(* CODESYS project Apollo_001_V1_CleanLease_Gemert_RECOVERED_2025-04-10T15-18-59.project

Project tree, tasks and I/O mapping:
  Device : CPX-E-CEC-M1-PN, Festo, order no. 4252743, version 3.5.16.46
    application Application
      libraries: Standard, 3.5.15.0 (System); CmpOPCUAClient, 3.5.17.0 (System); CmpOPCUAStack, 3.5.17.0 (System); IecVarAccessOpcUaMetaData Interfaces, * (System); CmpOPCUAServer Interfaces, * (System); Datasource OpcUa, * (3S - Smart Software Solutions GmbH); IecVarAccess3 Interfaces, * (System); SymbolicVarsBase, 3.5.16.30 (System); CmpBitmapPool, * (System)
      task MainTask (cyclic, interval t#20ms, priority 20) calls nothing
      task VISU_TASK (cyclic, interval 100 ms, priority 31) calls VisuElems.Visu_Prg
      task EtherCAT_Task (cyclic, interval t#8ms, priority 1) calls Apollo_Test_Mode, Apollo_Machine_State_V2, Set_Parameter_Prog, Test_Full_Prod, Dropconveyor
      program PLC_PRG [ST]
      image pool ImagePool
      Symbols
      Old_Progs/
        program Apollo_Machine_State [ST]
        function block FunctionBlock_Move_Guiders_Apollo [ST]
        program Apollo_Running_Guiders_AND_PickConveyor [ST]
        function block FunctionBlock_Move_Conveyor_Drop [ST]
        program Apollo_Running_GuiderMovement [ST]
      Progs_In_Apollo/
        Test_Mode/
          program Apollo_Test_Mode [ST]
          program Test_Full_Prod [ST]
        Machine State/
          program Set_Parameter_Prog [ST]
          program Apollo_Machine_State_V2 [ST]
        Run_Mode/
        FunctionBlocks/
          function block FunctionBlock_Gripper_Drop [ST]
          function block FunctionBlock_Move_To_Pos [ST]
          function block FunctionBlock_Gripper_Grip [ST]
          function block FunctionBlock_Activate_Ventilator [ST]
          function block FunctionBlock_Move_Pick_Conveyor [ST]
      visualisation Main_Page
      Variables_AND_Parameters/
        global variables Parameters
        global variables GVL_1
      Prog_In_DEV/
        Function Blocks/
        Programms/
          program Dropconveyor [ST]
          program Apollo_RunMode_Main [ST]
    SoftMotion General Axis Pool
    PLC_Diagnosis : PLC-Diagnosis, Festo AG & Co. KG, version 3.5.4.4
    CPX_E_System : CPX_E_System, Festo, order no. 4252743, version 1.311
      E_4AO_U_I : E-4AO-U-I, Festo, order no. 4080494, version 1.311
          settings:  = 0;  = 1;  = 1;  = 1;  = 1;  = 0;  = 0;  = 1;  = 144;  = 144;  = 144;  = 144;  = 1;  = 1;  = 1;  = 1;  = 0;  = 0;  = 0;  = 0;  = 0;  = 0;  = 0;  = 0;  = 0;  = 0;  = 0;  = 0;  = 0;  = 0;  = 0;  = 0;  = 0;  = 0;  = 0;  = 0;  = 0;  = 0;  = 0;  = 0;
             = 4466775293954;  = 'PI%i.0.1.1=1';  = 'PI%i.0.2.1=1';  = 'PI%i.0.7.1=1';  = 'PI%i.1.1.1=1';  = 'PI%i.1.3.1=0';  = 'PI%i.6.0.1=0';  = 'PI%i.6.5.1=1';  = 'PI%i.7.0.8=144';  = 'PI%i.8.0.8=144';  = 'PI%i.9.0.8=144';  = 'PI%i.10.0.8=144';  = 'PI%i.11.0.4=1';  = 'PI%i.11.4.4=1';  = 'PI%i.12.0.4=1';  = 'PI%i.12.4.4=1';  = dd8ed08c;  = 2
          output Application.GVL_1.Ventilator : UINT  // Output 0
          unmapped channels: Output 1, Output 2, Output 3
      E_8DO : E-8DO, Festo, order no. 4080491, version 1.311
          settings:  = 0;  = 1;  = 1;  = 0;  = 0;  = 0;  = 0;  = 0;  = 0;  = 0;  = 0;  = 0;  = 0;  = 0;  = 0;  = 0;  = 0;  = 0;  = 0;  = 0;  = 0;  = 0;  = 0;  = 0;  = 0;  = 0;  = 0;  = 0;  = 0;  = 0;  = 0;  = 0;  = 0;  = 0;  = 0;  = 0;  = 0;  = 0;  = 0;  = 0;
             = 0;  = 0;  = 0;  = 0;  = 0;  = 0;  = 0;  = 0;  = 0;  = 0;  = 0;  = 0;  = 8800390021120;  = 'PI%i.0.1.1=1';  = 'PI%i.0.2.1=1';  = 'PI%i.1.1.1=0';  = dd8aeb00;  = 1
          output Application.GVL_1.Conveyor_Pick_Speed_A : BOOL  // Output 0.Bit0
          output Application.GVL_1.Conveyor_Pick_Speed_B : BOOL  // Output 0.Bit1
          output Application.GVL_1.Conveyor_Pick_Speed_C : BOOL  // Output 0.Bit2
          output Application.GVL_1.Conveyor_Pick_Reverse : BOOL  // Output 0.Bit3
          output Application.GVL_1.Conveyor_Drop_Speed_A : BOOL  // Output 0.Bit4
          output Application.GVL_1.Conveyor_Drop_Speed_B : BOOL  // Output 0.Bit5
          output Application.GVL_1.Conveyor_Drop_Speed_C : BOOL  // Output 0.Bit6
          output Application.GVL_1.Conveyor_Drop_Reverse : BOOL  // Output 0.Bit7
          unmapped channels: Output 0
      E_8DO_1 : E-8DO, Festo, order no. 4080491, version 1.311
          settings:  = 0;  = 1;  = 1;  = 0;  = 0;  = 0;  = 0;  = 0;  = 0;  = 0;  = 0;  = 0;  = 0;  = 0;  = 0;  = 0;  = 0;  = 0;  = 0;  = 0;  = 0;  = 0;  = 0;  = 0;  = 0;  = 0;  = 0;  = 0;  = 0;  = 0;  = 0;  = 0;  = 0;  = 0;  = 0;  = 0;  = 0;  = 0;  = 0;  = 0;
             = 0;  = 0;  = 0;  = 0;  = 0;  = 0;  = 0;  = 0;  = 0;  = 0;  = 0;  = 0;  = 8800390021120;  = 'PI%i.0.1.1=1';  = 'PI%i.0.2.1=1';  = 'PI%i.1.1.1=0';  = dd8b5e24;  = 1
          output Application.GVL_1.Gripper : BOOL  // Output 0.Bit0
          output Application.GVL_1.Blow_Out : BOOL  // Output 0.Bit1
          output Application.GVL_1.VacuumBlow : BOOL  // Output 0.Bit2
          unmapped channels: Output 0
      E_16DI : E-16DI, Festo, order no. 4080492, version 1.311
          settings:  = 0;  = 1;  = 1;  = 1;  = 1;  = 0;  = 0;  = 0;  = 0;  = 0;  = 0;  = 0;  = 0;  = 0;  = 0;  = 0;  = 0;  = 0;  = 0;  = 0;  = 0;  = 0;  = 0;  = 0;  = 0;  = 0;  = 0;  = 0;  = 0;  = 0;  = 0;  = 0;  = 0;  = 0;  = 0;  = 0;  = 0;  = 0;  = 0;  = 0;
             = 0;  = 0;  = 0;  = 0;  = 0;  = 0;  = 0;  = 0;  = 0;  = 0;  = 0;  = 0;  = 0;  = 1153202979585458176;  = 'PI%i.0.0.1=1';  = 'PI%i.1.0.1=1';  = 'PI%i.1.4.2=1';  = 'PI%i.1.6.2=1';  = 'PI%i.6.0.1=0';  = 'PI%i.6.1.1=0';  = 'PI%i.6.2.1=0';  = 'PI%i.6.3.1=0';  = 'PI%i.6.4.1=0';  = 'PI%i.6.5.1=0';  = 'PI%i.6.6.1=0';  = 'PI%i.6.7.1=0';  = 'PI%i.7.0.1=0';  = 'PI%i.7.1.1=0';  = 'PI%i.7.2.1=0';  = 'PI%i.7.3.1=0';  = 'PI%i.7.4.1=0';  = 'PI%i.7.5.1=0';  = 'PI%i.7.6.1=0';  = 'PI%i.7.7.1=0';  = dd8b6c92;  = 1
          input  Application.GVL_1.PHC_PickConveyor_END : BOOL  // Input 0.Bit0
          input  Application.GVL_1.Start_production_Button : BOOL  // Input 0.Bit2
          input  Application.GVL_1.PHC_Drop_Conveyor : BOOL  // Input 0.Bit6
          unmapped channels: Input 0
      E_CEC_M1_PN : E-CEC-M1-PN, Festo, order no. 4252743, version 1.311
          settings:  = 0;  = 15365580000768;  = 16820416;  = 16777215;  = 0;  = 14549093;  = 1f93f90d;  = 11
    PROFINET_Device : PROFINET Device, Festo, version 3.5.15.2
    EtherCAT_Master : EtherCAT Master, Festo, version 3.5.16.43
      CMMT_AS_MP_S1 : CMMT-AS-MP-S1 (SoftMotion), Festo, order no. 814316x, version 4.0.33.0
          settings: StationAlias = 0
          unmapped channels: Controlword, Modes of operation, Target position, Profile velocity, Target velocity, Target torque, Velocity offset, Torque offset, Touch probe function, ---, Statusword, Modes of operation display, Position actual value, Velocity actual value, Torque actual value, Touch probe status, Touch probe 1 positive edge, Touch probe 1 negative edge, Touch probe 2 positive edge, Touch probe 2 negative edge, ---
        Inner_Rail : SM_Drive_EtherCAT_Festo_CMMT_AS_MP_S1, Festo, version 4.0.33.0
            settings: wDriveID = 0; fSWLimitPositive = 1400; fSWLimitNegative = -50; AdrOffset_8010 = 12; BitOffset_8010 = 0; BitLength_8010 = 16; Address_8010 = '%QW6'; Type_8010 = 'UINT'; AddressPointer_8010 = ADR(%QW6); AdrOffset_8020 = 14; BitOffset_8020 = 0; BitLength_8020 = 8; Address_8020 = '%QB14'; Type_8020 = 'SINT'; AddressPointer_8020 = ADR(%QB14); AdrOffset_8030 = 16; BitOffset_8030 = 0; BitLength_8030 = 32; Address_8030 = '%QD4'; Type_8030 = 'DINT'; AddressPointer_8030 = ADR(%QD4); AdrOffset_8040 = 24; BitOffset_8040 = 0; BitLength_8040 = 32; Address_8040 = '%QD6'; Type_8040 = 'DINT'; AddressPointer_8040 = ADR(%QD6); AdrOffset_8050 = 28; BitOffset_8050 = 0; BitLength_8050 = 16; Address_8050 = '%QW14'; Type_8050 = 'INT'; AddressPointer_8050 = ADR(%QW14); AdrOffset_8060 = 38; BitOffset_8060 = 0; BitLength_8060 = 16; Address_8060 = '%QW19'; Type_8060 = 'UINT'; AddressPointer_8060 = ADR(%QW19); AdrOffset_8510 = 4;
              BitOffset_8510 = 0; BitLength_8510 = 16; Address_8510 = '%IW2'; Type_8510 = 'UINT'; AddressPointer_8510 = ADR(%IW2); AdrOffset_8520 = 6; BitOffset_8520 = 0; BitLength_8520 = 8; Address_8520 = '%IB6'; Type_8520 = 'SINT'; AddressPointer_8520 = ADR(%IB6); AdrOffset_8530 = 8; BitOffset_8530 = 0; BitLength_8530 = 32; Address_8530 = '%ID2'; Type_8530 = 'DINT'; AddressPointer_8530 = ADR(%ID2); AdrOffset_8540 = 12; BitOffset_8540 = 0; BitLength_8540 = 32; Address_8540 = '%ID3'; Type_8540 = 'DINT'; AddressPointer_8540 = ADR(%ID3); AdrOffset_8550 = 16; BitOffset_8550 = 0; BitLength_8550 = 16; Address_8550 = '%IW8'; Type_8550 = 'INT'; AddressPointer_8550 = ADR(%IW8); AdrOffset_8560 = 18; BitOffset_8560 = 0; BitLength_8560 = 16; Address_8560 = '%IW9'; Type_8560 = 'UINT'; AddressPointer_8560 = ADR(%IW9); AdrOffset_8570 = 20; BitOffset_8570 = 0; BitLength_8570 = 32; Address_8570 = '%ID5'; Type_8570 = 'DINT';
              AddressPointer_8570 = ADR(%ID5); AdrOffset_8580 = 24; BitOffset_8580 = 0; BitLength_8580 = 32; Address_8580 = '%ID6'; Type_8580 = 'DINT'; AddressPointer_8580 = ADR(%ID6); AdrOffset_8590 = 28; BitOffset_8590 = 0; BitLength_8590 = 32; Address_8590 = '%ID7'; Type_8590 = 'DINT'; AddressPointer_8590 = ADR(%ID7); AdrOffset_8600 = 32; BitOffset_8600 = 0; BitLength_8600 = 32; Address_8600 = '%ID8'; Type_8600 = 'DINT'; AddressPointer_8600 = ADR(%ID8)
      CMMT_AS_MP_S1_1 : CMMT-AS-MP-S1 (SoftMotion), Festo, order no. 814316x, version 4.0.33.0
          settings: StationAlias = 0
          unmapped channels: Controlword, Modes of operation, Target position, Profile velocity, Target velocity, Target torque, Velocity offset, Torque offset, Touch probe function, ---, Statusword, Modes of operation display, Position actual value, Velocity actual value, Torque actual value, Touch probe status, Touch probe 1 positive edge, Touch probe 1 negative edge, Touch probe 2 positive edge, Touch probe 2 negative edge, ---
        Outer_Rail : SM_Drive_EtherCAT_Festo_CMMT_AS_MP_S1, Festo, version 4.0.33.0
            settings: fSWLimitPositive = 1400; fSWLimitNegative = -50; AdrOffset_8010 = 44; BitOffset_8010 = 0; BitLength_8010 = 16; Address_8010 = '%QW22'; Type_8010 = 'UINT'; AddressPointer_8010 = ADR(%QW22); AdrOffset_8020 = 46; BitOffset_8020 = 0; BitLength_8020 = 8; Address_8020 = '%QB46'; Type_8020 = 'SINT'; AddressPointer_8020 = ADR(%QB46); AdrOffset_8030 = 48; BitOffset_8030 = 0; BitLength_8030 = 32; Address_8030 = '%QD12'; Type_8030 = 'DINT'; AddressPointer_8030 = ADR(%QD12); AdrOffset_8040 = 56; BitOffset_8040 = 0; BitLength_8040 = 32; Address_8040 = '%QD14'; Type_8040 = 'DINT'; AddressPointer_8040 = ADR(%QD14); AdrOffset_8050 = 60; BitOffset_8050 = 0; BitLength_8050 = 16; Address_8050 = '%QW30'; Type_8050 = 'INT'; AddressPointer_8050 = ADR(%QW30); AdrOffset_8060 = 70; BitOffset_8060 = 0; BitLength_8060 = 16; Address_8060 = '%QW35'; Type_8060 = 'UINT'; AddressPointer_8060 = ADR(%QW35); AdrOffset_8510 = 40; BitOffset_8510 = 0;
              BitLength_8510 = 16; Address_8510 = '%IW20'; Type_8510 = 'UINT'; AddressPointer_8510 = ADR(%IW20); AdrOffset_8520 = 42; BitOffset_8520 = 0; BitLength_8520 = 8; Address_8520 = '%IB42'; Type_8520 = 'SINT'; AddressPointer_8520 = ADR(%IB42); AdrOffset_8530 = 44; BitOffset_8530 = 0; BitLength_8530 = 32; Address_8530 = '%ID11'; Type_8530 = 'DINT'; AddressPointer_8530 = ADR(%ID11); AdrOffset_8540 = 48; BitOffset_8540 = 0; BitLength_8540 = 32; Address_8540 = '%ID12'; Type_8540 = 'DINT'; AddressPointer_8540 = ADR(%ID12); AdrOffset_8550 = 52; BitOffset_8550 = 0; BitLength_8550 = 16; Address_8550 = '%IW26'; Type_8550 = 'INT'; AddressPointer_8550 = ADR(%IW26); AdrOffset_8560 = 54; BitOffset_8560 = 0; BitLength_8560 = 16; Address_8560 = '%IW27'; Type_8560 = 'UINT'; AddressPointer_8560 = ADR(%IW27); AdrOffset_8570 = 56; BitOffset_8570 = 0; BitLength_8570 = 32; Address_8570 = '%ID14'; Type_8570 = 'DINT'; AddressPointer_8570 = ADR(%ID14);
              AdrOffset_8580 = 60; BitOffset_8580 = 0; BitLength_8580 = 32; Address_8580 = '%ID15'; Type_8580 = 'DINT'; AddressPointer_8580 = ADR(%ID15); AdrOffset_8590 = 64; BitOffset_8590 = 0; BitLength_8590 = 32; Address_8590 = '%ID16'; Type_8590 = 'DINT'; AddressPointer_8590 = ADR(%ID16); AdrOffset_8600 = 68; BitOffset_8600 = 0; BitLength_8600 = 32; Address_8600 = '%ID17'; Type_8600 = 'DINT'; AddressPointer_8600 = ADR(%ID17)
  libraries: VisuSymbols, 4.5.0.0 (System)
  5ce3da45-db07-42e7-a21c-a00fff4ed8f6|C:\Users\RobinvanNieuwenhuyse\Downloads\Landuwasco-logo.png
  text list GlobalTextList
*)

// Device/Application/Variables_AND_Parameters/Parameters
{attribute 'qualified_only'}
VAR_GLOBAL PERSISTENT RETAIN
//-------------------------------------------------------------------------------------------------
//Positions
	//Readypos
	ReadyPos_Inner:INT;
	ReadyPos_Outer:INT;
	
	//Pick_Pos
	Pick_Pos_Inner_Test_Prod:INT;
	Pick_Pos_Outer_Test_Prod:INT;
	
	//Drop_Pos
	Drop_Pos_Inner:INT;
	Drop_Pos_Outer:INT;
	
	Drop_Pos_Inner_Test_Prod:INT;
	Drop_Pos_Outer_Test_Prod:INT;
	
	//Before Drop Pos
	Before_Drop_Pos_Inner:INT;
	Before_Drop_Pos_Outer:INT;
	
	//Distances
	Distance_Move_After_PHC:LREAL; // distance in mm
	
	
	//Points between readypos and Pick_Pos called RPP_CheckPointPos
	
//-------------------------------------------------------------------------------------------------
//Dynamics
	//Test 
	Speed_Test_Prod:LREAL; // for the test production cycly
	ACC_DEC_Test_Prod:LREAl;
	Jerk_Test_Prod:LREAL;
	
	Speed_Test_Prod_Slow:LREAL;
	ACC_DEC_Test_Prod_Slow:LREAL;
	Jerk_Test_prod_Slow:LREAL;
	
	//Production
	Vel_Prod:LREAL;
	Acc_Dec_Prod:LREAL;
	Jerk_Prod:LREAL;
//-------------------------------------------------------------------------------------------------
//Timers

//Wait times
	Wait_Time_NoBatch:INT;	
	Wait_Time_Piece_Drop_Conveyor:INT;// max time the drop conveyor can run (if no pieces are detected
	Wait_Time_AI:INT;
	
//Delays
	Delay_Gripper_Closed_Before_Moving:INT;
	Delay_Move_After_Piece_Dropped:INT;
	Delay_Blow_Vacuum:INT;
	Delay_Move_Conveyor_After_PHC_Covered:INT;
	Delay_DropBox_Opened:INT;
	Delay_Conveyor_Move_After_DropBox_Opened:INT;
	Delay_Gripper_Open_During_Drop:INT;
//-------------------------------------------------------------------------------------------------
// Settings
	//Ventilator
	Ventilator_Strength:INT;	

	//Conveyors
	Conveyor_Speed_Pick:INT;	
	Conveyor_Speed_Drop:INT;		

	Delay_Blow:INT;

END_VAR

// Device/Application/Variables_AND_Parameters/GVL_1
{attribute 'qualified_only'}
VAR_GLOBAL
//-------------------------------------------------------------------------------------------------	
// AI 
	//States
	AI_Start:BOOL;
	AI_Done:BOOL;
	AI_Detection_Memory:BOOL;
	
	AI_USE_TestProd:BOOL;
	
	//Detections
	Pick_Pos_Inner:INT;
	Pick_Pos_Outer:INT;
	
	Conveyor_Pick_Move_Left:BOOL;
	Conveyor_Pick_Move_Right:BOOL;
	Conveyor_Pick_Time:INT; // Time in ms for movement left or right
	Conveyor_Movement_Memory:BOOL; // check if conveyor already moved due to detections before
//-------------------------------------------------------------------------------------------------		
// Robot Command Settings

	//Power Drives
	Power_Drive_InnerRail:MC_Power;
	Power_Drive_OuterRail:MC_Power;
	
	//Reset
	Reset_InnerRail:MC_Reset;
	Reset_OuterRail:MC_Reset;
	
	//movements 
	Move_To_Pos_InnerRail:MC_MoveAbsolute;
	Move_To_Pos_OuterRail:MC_MoveAbsolute;
	
	//Stop movement and set axis in standstill
	Halt_Inner:MC_Halt;
	Halt_Outer:MC_Halt;
//-------------------------------------------------------------------------------------------------		
//	Buttons
	Turn_On:BOOL; // OPCUA communicated
	Turn_Off:BOOL; // OPCUA communicated
	Reset:BOOL;
	Start_production_Button:BOOL;
//-------------------------------------------------------------------------------------------------	
//Sensors
	//PHC
	PHC_PickConveyor_Front:BOOL; //first PHC in cycle picking
	PHC_PickConveyor_END:BOOL;  // last PHC
	
	
	PHC_Reach_Batch:BOOL;
	PHC_Drop_Conveyor:BOOL;
	PHC_Gripper:BOOL;
//-------------------------------------------------------------------------------------------------	
//Actuators

	//Conveyors
	Conveyor_Pick_Speed_A:BOOL;
	Conveyor_Pick_Speed_B:BOOL;
	Conveyor_Pick_Speed_C:BOOL;
	Conveyor_Pick_Reverse:BOOL;
	Test_Conveyor_Pick_Choose_Speed:INT:=1;
	
	Conveyor_Drop_Speed_A:BOOL;
	Conveyor_Drop_Speed_B:BOOL;
	Conveyor_Drop_Speed_C:BOOL;
	Conveyor_Drop_Reverse:BOOL;
	Test_coveyor_Drop_Choos_Speed:INT:=1;
	
	//Gripper
	Gripper:BOOL;
	VacuumBlow:BOOL;
	Blow_Out:BOOL;
	
	//Ventilator
	Ventilator:INT;
	
	//DropBox
	Cylinder_DropBox:BOOL;
	
//-------------------------------------------------------------------------------------------------	
// State of Robot
//Positions
	//Current Pos
	Current_Pos_Inner:LREAL;
	Current_Pos_Outer:LREAL;
// Cases of Robot
	//Test
	enStepTestProd:INT; // this variable is purely to test prod during dev
	enStepTest:INT; //case for testmode

	
	//Prod
	enStepBoot:INT; // case int for bootup proces
	enStepRun:INT; // case int for when robot is running
	enStepRunMove:INT; //case int for moving robot
	enStepDrop:INT;
	
//Cases of Functions
	enFBMoveGuider:INT; // case int for certain movements
	enFBMoveConveyor_Pick:INT;
	enFBMoveConveyor_Drop:INT;
	enFBGripping:INT;
	enFBDropping:INT;
	enFBMove_To_Pos:INT;
	enFBVentilator:INT;
	
	
	
//Cases of methods
	enMeCheckStateBatch:INT;
	
//States of robot
	//prod
	Machine_In_Error:BOOL;
	Machine_Ready_To_Run:BOOL;
	Machine_Production_Mode:BOOL;
	
	//test
	Machine_Test_Mode:BOOL;
	Machine_TestProd_Mode:BOOL; // OPCUA communicated

//States of production
	BatchOnPickConveyor:BOOL; // Check if batch is on Conveyor
	PutinBatch:BOOL; // start signal if batch is put in the robot
	PieceOnDropConveyor:BOOL;

//Test functions
	Test_Move:BOOL; // This initiates a Test_Move
	Test_Pick_Conveyor:BOOL; // this initiates single move for 
	Test_Ventilator:BOOL;
	Test_Drop_Conveyor:BOOL;
	
	Test_Time_Move_Pick_Conveyor:INT:=1000; // for testmode
	Test_Pick_Conveyor_Left:BOOL:=FALSE; // for testmode
	Test_Pick_Conveyor_Right:BOOL:=TRUE; // for testmode
	
	Test_Drop_Conveyor_Forward:BOOL:=TRUE;
	Test_Drop_Conveyor_Backward:BOOL;
	
	
//-------------------------------------------------------------------------------------------------	
//positions

	//Test values Positions
	Test_Pos_Inner_Rail:LREAL:=1020;
	Test_Pos_Outer_Rail:LREAL:=1150;

	//Max positions
	Max_Diff_Inner_Outer:INT:=250; // onder under low positions
	Min_Diff_Inner_Outer:INT:=10;

	//Max positions to pick
	Max_Pick_Inner:LREAL; // max position Inner
	Max_Pick_Outer:LREAL; // max position outer
//-------------------------------------------------------------------------------------------------	
//Dynamics

	//Test values Dynamics
	Test_Vel:INT:=30;
	Test_Acc_Dec:INT:=1000;
	Test_Jerk:LREAL:=100000;
	
	
//-------------------------------------------------------------------------------------------------	
//Parameters
	Set_Parameters_Default:BOOL;

	




END_VAR

// Device/Application/Progs_In_Apollo/Test_Mode/Apollo_Test_Mode
PROGRAM Apollo_Test_Mode
VAR
	FB_Conveyor_Pick_Move:FunctionBlock_Move_Pick_Conveyor;
	FB_Move_To_Pos:FunctionBlock_Move_To_Pos;
	FB_Ventilator:FunctionBlock_Activate_Ventilator;
END_VAR

CASE GVL_1.enStepTest OF
	0: // Wait Until test_Mode is activated and reset all function POU
		IF GVL_1.Machine_Ready_To_Run AND GVL_1.Machine_Test_Mode THEN
					//Setup settings for axis:
					
					
					
			GVL_1.Move_To_Pos_InnerRail.Velocity:=GVL_1.Test_Vel;
			GVL_1.Move_To_Pos_InnerRail.Acceleration:=GVL_1.Test_Acc_Dec;
			GVL_1.Move_To_Pos_InnerRail.Deceleration:=GVL_1.Test_Acc_Dec;
			GVL_1.Move_To_Pos_InnerRail.Jerk:=GVL_1.Test_Jerk;
			
			GVL_1.Move_To_Pos_OuterRail.Velocity:=GVL_1.Test_Vel;
			GVL_1.Move_To_Pos_OuterRail.Acceleration:=GVL_1.Test_Acc_Dec;
			
			GVL_1.Move_To_Pos_OuterRail.Deceleration:=GVL_1.Test_Acc_Dec;
			GVL_1.Move_To_Pos_OuterRail.Jerk:=GVL_1.Test_Jerk;
			
			GVL_1.enStepTest:=GVL_1.enStepTest+10;
		END_IF
		

		
		
		
	10: // Decide what will be tested
		IF GVL_1.Test_Move THEN
			GVL_1.enStepTest:=20;
		END_IF
		
		IF GVL_1.Test_Pick_Conveyor THEN
			GVL_1.enStepTest:=30;
		END_IF
		
		
		IF GVL_1.Test_Ventilator THEN
			FB_Ventilator(Start:=TRUE);
		ELSE
			FB_Ventilator(Start:=FALSE);
		END_IF
		
		
		
	20:// Test a single move guiders
		
		FB_Move_To_Pos(Start:=TRUE,Position_Inner:=GVL_1.Test_Pos_Inner_Rail,Position_Outer:=GVL_1.Test_Pos_Outer_Rail);
		
		IF FB_Move_To_Pos.Done THEN
			GVL_1.Test_Move:=FALSE;
			FB_Move_To_Pos(Start:=FALSE,Position_Inner:=GVL_1.Test_Pos_Inner_Rail,Position_Outer:=GVL_1.Test_Pos_Outer_Rail);
			GVL_1.enStepTest:=100;
		END_IF
		

		
	30:// test a single move pick coveyor
		FB_Conveyor_Pick_Move(Time_Moving:=GVL_1.Test_Time_Move_Pick_Conveyor,Left:=GVL_1.Test_Pick_Conveyor_Left,Right:=GVL_1.Test_Pick_Conveyor_Right,Speed:=GVL_1.Test_Conveyor_Pick_Choose_Speed,Start:=TRUE);
		
		IF FB_Conveyor_Pick_Move.Done THEN
			FB_Conveyor_Pick_Move(Time_Moving:=GVL_1.Test_Time_Move_Pick_Conveyor,Left:=GVL_1.Test_Pick_Conveyor_Left,Right:=GVL_1.Test_Pick_Conveyor_Right,Start:=FALSE);
			GVL_1.Test_Pick_Conveyor:=FALSE;
			GVL_1.enStepTest:=100;
		END_IF
		
	
	100: // Reset and go back to start
		GVL_1.Move_To_Pos_InnerRail(Axis:=Inner_Rail, Position:=GVL_1.Test_Pos_Inner_Rail,Execute:=FALSE);
		GVL_1.Move_To_Pos_OuterRail(Axis:=Outer_Rail, Position:=GVL_1.Test_Pos_Outer_Rail,Execute:=FALSE);
		
		
		GVL_1.enStepTest:=0;
		
	
END_CASE

IF NOT GVL_1.Machine_Test_Mode THEN
	GVL_1.enStepTest:=0;
END_IF

END_PROGRAM

// Device/Application/Progs_In_Apollo/FunctionBlocks/FunctionBlock_Move_Pick_Conveyor
FUNCTION_BLOCK FunctionBlock_Move_Pick_Conveyor
VAR_INPUT
	Time_Moving:INT;
	Left:BOOL;
	Right:BOOL;
	Speed:INT;
	Start:BOOL;
END_VAR
VAR_OUTPUT
	Done:BOOL;
END_VAR
VAR
	Timer:TON;
END_VAR

CASE GVL_1.enFBMoveConveyor_Pick OF
	0:// Wait until Start
		IF Start AND NOT Done THEN
			GVL_1.enFBMoveConveyor_Pick:=GVL_1.enFBMoveConveyor_Pick+10;
		END_IF
		
		IF NOT Start THEN
			Done:=FALSE;
		END_IF
	10: // Move conveyor in correct direction for the time needed to move
		IF Speed = 1 THEN
			GVL_1.Conveyor_Pick_Speed_C:=TRUE;
		ELSIF Speed = 2 THEN
			GVL_1.Conveyor_Pick_Speed_B:=TRUE;
		ELSIF Speed=3 THEN
			GVL_1.Conveyor_Pick_Speed_A:=TRUE;
		ELSIF Speed = 4 THEN
			GVL_1.Conveyor_Pick_Speed_C:=TRUE;
			GVL_1.Conveyor_Pick_Speed_B:=TRUE;
		ELSIF Speed = 5 THEN
			GVL_1.Conveyor_Pick_Speed_A:=TRUE;
			GVL_1.Conveyor_Pick_Speed_B:=TRUE;
			GVL_1.Conveyor_Pick_Speed_C:=TRUE;
		ELSE
			GVL_1.enFBMoveConveyor_Pick:=GVL_1.enFBMoveConveyor_Pick+10;
		END_IF
		
		IF Left THEN
			GVL_1.Conveyor_Pick_Reverse:=FALSE;
		ELSE
			GVL_1.Conveyor_Pick_Reverse:=TRUE;
		END_IF
		
		Timer(In:=TRUE,PT:=INT_TO_TIME(Time_Moving));
		
		IF Timer.Q OR NOT Start THEN
			GVL_1.enFBMoveConveyor_Pick:=GVL_1.enFBMoveConveyor_Pick+10;
		END_IF



	20:// reset
		GVL_1.Conveyor_Pick_Speed_A:=FALSE;
		GVL_1.Conveyor_Pick_Speed_B:=FALSE;
		GVL_1.Conveyor_Pick_Speed_C:=FALSE;
		Timer(IN:=FALSE);
		Done:=TRUE;
		
		GVL_1.enFBMoveConveyor_Pick:=0;
END_CASE

END_FUNCTION_BLOCK

// Device/Application/Progs_In_Apollo/FunctionBlocks/FunctionBlock_Move_To_Pos
FUNCTION_BLOCK FunctionBlock_Move_To_Pos
VAR_INPUT
	Start:BOOL;
	Position_Inner:LREAL;
	Position_Outer:LREAL;
	Halt:BOOL;
END_VAR
VAR_OUTPUT
	Done:BOOL;
END_VAR
VAR
	dx_Inner:LREAL;
	dx_Outer:LREAL;
	v_Inner:LREAL;
END_VAR

CASE GVL_1.enFBMove_To_Pos OF
	0:// wait until init
		
		IF NOT Start THEN
			Done:=FALSE;
			Halt:=FALSE;
		END_IF
		
		
		IF Start AND NOT Done AND NOT GVL_1.Machine_In_Error AND NOT Halt THEN
			GVL_1.enFBMove_To_Pos:=GVL_1.enFBMove_To_Pos+10;
		END_IF
		
	10: // Set all necesarry settings 
		GVL_1.Move_To_Pos_OuterRail.Position:=Position_Outer;
		GVL_1.Move_To_Pos_InnerRail.Position:=Position_Inner;
		
		dx_Inner:=ABS(GVL_1.Current_Pos_Inner-Position_Inner);
		dx_Outer:=ABS(GVL_1.Current_Pos_Outer-Position_Outer);
		
		IF dx_Outer <= 100 or dx_Inner <= 100 THEN
			v_Inner:=GVL_1.Move_To_Pos_OuterRail.Velocity;
		ELSE
			v_Inner:=((GVL_1.Move_To_Pos_OuterRail.Velocity)*(dx_Inner))/(dx_Outer);
		END_IF

		GVL_1.Move_To_Pos_InnerRail.Velocity:= v_Inner;
		
		
		
		GVL_1.enFBMove_To_Pos:=GVL_1.enFBMove_To_Pos+10;
	20: // do move

		GVL_1.Move_To_Pos_InnerRail(Axis:=Inner_Rail,Execute:=TRUE);
		GVL_1.Move_To_Pos_OuterRail(Axis:=Outer_Rail,Execute:=TRUE);

		IF Halt THEN
			GVL_1.Move_To_Pos_InnerRail(Axis:=Inner_Rail,Execute:=FALSE);
			GVL_1.Move_To_Pos_OuterRail(Axis:=Outer_Rail,Execute:=FALSE);
			GVL_1.enFBMove_To_Pos:=GVL_1.enFBMove_To_Pos+10;
		END_IF		

		IF GVL_1.Move_To_Pos_InnerRail.Done AND GVL_1.Move_To_Pos_OuterRail.Done THEN
			GVL_1.Move_To_Pos_InnerRail(Axis:=Inner_Rail,Execute:=FALSE);
			GVL_1.Move_To_Pos_OuterRail(Axis:=Outer_Rail,Execute:=FALSE);
			Done:=TRUE;
			GVL_1.enFBMove_To_Pos:=0;
		END_IF
	30: // execute Halt
		GVL_1.Halt_Inner(Axis:=Inner_Rail,Deceleration:=GVL_1.Move_To_Pos_InnerRail.Deceleration,Jerk:=GVL_1.Move_To_Pos_InnerRail.Jerk,Execute:=TRUE);
		GVL_1.Halt_Outer(Axis:=Outer_Rail,Deceleration:=GVL_1.Move_To_Pos_OuterRail.Deceleration,Jerk:=GVL_1.Move_To_Pos_OuterRail.Jerk,Execute:=TRUE);
		
		IF GVL_1.Halt_Inner.Done AND GVL_1.Halt_Outer.Done THEN
			GVL_1.Move_To_Pos_InnerRail(Axis:=Inner_Rail,Execute:=FALSE);
			GVL_1.Move_To_Pos_OuterRail(Axis:=Outer_Rail,Execute:=FALSE);
			
			GVL_1.Halt_Inner(Axis:=Inner_Rail,Execute:=FALSE);
			GVL_1.Halt_Outer(Axis:=Outer_Rail,Execute:=FALSE);
			
			GVL_1.enFBMove_To_Pos:=GVL_1.enFBMove_To_Pos+10;
		END_IF
	40: // move distance after a halt
		GVL_1.Move_To_Pos_InnerRail(Axis:=Inner_Rail,Position:=(GVL_1.Current_Pos_Inner-Parameters.Distance_Move_After_PHC),Execute:=TRUE);
		GVL_1.Move_To_Pos_OuterRail(Axis:=Outer_Rail,Position:=(GVL_1.Current_Pos_Outer-Parameters.Distance_Move_After_PHC),Execute:=TRUE);
		
		IF GVL_1.Move_To_Pos_InnerRail.Done AND GVL_1.Move_To_Pos_OuterRail.Done THEN
			GVL_1.Move_To_Pos_InnerRail(Axis:=Inner_Rail,Execute:=FALSE);
			GVL_1.Move_To_Pos_OuterRail(Axis:=Outer_Rail,Execute:=FALSE);
			
			Done:=TRUE;
			
			
			GVL_1.enFBMove_To_Pos:=0;
		END_IF
		
		
END_CASE

END_FUNCTION_BLOCK

// Device/Application/Progs_In_Apollo/FunctionBlocks/FunctionBlock_Activate_Ventilator
FUNCTION_BLOCK FunctionBlock_Activate_Ventilator
VAR_INPUT
	Start:BOOL;
END_VAR
VAR_OUTPUT
END_VAR
VAR
END_VAR

CASE GVL_1.enFBVentilator OF
	0:// wait until Start
		IF Start THEN
			GVL_1.enFBVentilator:=GVL_1.enFBVentilator+10;
		END_IF
	10:// Turn on Ventilator
		GVL_1.Ventilator:=Parameters.Ventilator_Strength;
		
		IF NOT Start THEN
			GVL_1.Ventilator:=0;
			GVL_1.enFBVentilator:=0;
		END_IF
END_CASE

END_FUNCTION_BLOCK

// Device/Application/Progs_In_Apollo/Machine State/Apollo_Machine_State_V2
PROGRAM Apollo_Machine_State_V2
VAR
END_VAR

CASE GVL_1.enStepBoot OF
	0:// Wait until Init 
		IF NOT GVL_1.Machine_In_Error AND GVL_1.Turn_On THEN
			GVL_1.Turn_Off:=FALSE;
			GVL_1.enStepBoot:=GVL_1.enStepBoot+10;
		END_IF
	
	10://Boot up drive
		GVL_1.Power_Drive_InnerRail(Axis:=Inner_Rail,Enable:=TRUE,bRegulatorOn:=TRUE,bDriveStart:=TRUE);
		GVL_1.Power_Drive_OuterRail(Axis:=Outer_Rail,Enable:=TRUE,bRegulatorOn:=TRUE,bDriveStart:=TRUE);
		
		IF GVL_1.Power_Drive_InnerRail.Status AND GVL_1.Power_Drive_OuterRail.Status THEN
			GVL_1.Machine_Ready_To_Run:=TRUE;
			GVL_1.enStepBoot:=GVL_1.enStepBoot+10;
		END_IF
	20: // Power_On mode
		IF GVL_1.Move_To_Pos_InnerRail.Error OR GVL_1.Move_To_Pos_OuterRail.Error THEN
			GVL_1.Machine_Ready_To_Run:=FALSE;
			GVL_1.Machine_Test_Mode:=FALSE;
			GVL_1.Machine_TestProd_Mode:=FALSE;
			GVL_1.Turn_On:=FALSE;
			GVL_1.Machine_In_Error:=TRUE;
			
			
			GVL_1.enStepTest:=0;
			GVL_1.enStepTestProd:=0;
			
			GVL_1.enFBMove_To_Pos:=0;
			
			GVL_1.Power_Drive_InnerRail(Axis:=Inner_Rail,Enable:=FALSE,bRegulatorOn:=FALSE,bDriveStart:=FALSE);
			GVL_1.Power_Drive_OuterRail(Axis:=Outer_Rail,Enable:=FALSE,bRegulatorOn:=FALSE,bDriveStart:=FALSE);
			
			GVL_1.Move_To_Pos_InnerRail(Axis:=Inner_Rail,Execute:=FALSE);
			GVL_1.Move_To_Pos_OuterRail(Axis:=Outer_Rail,Execute:=FALSE);
			
			Inner_Rail.bRegulatorOn:=FALSE;
			Inner_Rail.bDriveStart:=FALSE;
			Outer_Rail.bRegulatorOn:=FALSE;
			Outer_Rail.bDriveStart:=FALSE;
			
			
			
			GVL_1.enStepBoot:=100;
		END_IF
		
		IF GVL_1.Turn_Off THEN
			GVL_1.Turn_On:=FALSE;
			GVL_1.Machine_Ready_To_Run:=FALSE;
			GVL_1.Machine_Test_Mode:=FALSE;
			
			GVL_1.Power_Drive_InnerRail(Axis:=Inner_Rail,Enable:=FALSE,bRegulatorOn:=FALSE,bDriveStart:=FALSE);
			GVL_1.Power_Drive_OuterRail(Axis:=Outer_Rail,Enable:=FALSE,bRegulatorOn:=FALSE,bDriveStart:=FALSE);
			
			Inner_Rail.bRegulatorOn:=FALSE;
			Inner_Rail.bDriveStart:=FALSE;
			Outer_Rail.bRegulatorOn:=FALSE;
			Outer_Rail.bDriveStart:=FALSE;
			
			
			
			GVL_1.enStepBoot:=0;
		END_IF
	
	
	100:// Errormode
    	IF GVL_1.Reset THEN
        // Reset InnerRail if in error
        	IF GVL_1.Move_To_Pos_InnerRail.Error THEN
            	GVL_1.Reset_InnerRail(Axis := Inner_Rail, Execute := TRUE);
        	END_IF
        
        // Reset OuterRail if in error
        	IF GVL_1.Move_To_Pos_OuterRail.Error THEN
            	GVL_1.Reset_OuterRail(Axis := Outer_Rail, Execute := TRUE);
        	END_IF

        // Check if both resets are done
        	IF GVL_1.Reset_InnerRail.Done THEN
            	GVL_1.Reset_InnerRail(Axis := Inner_Rail, Execute := FALSE);
        	END_IF
        
        	IF GVL_1.Reset_OuterRail.Done THEN
            	GVL_1.Reset_OuterRail(Axis := Outer_Rail, Execute := FALSE);
        	END_IF

        // When both are done, exit error mode
			IF (NOT GVL_1.Move_To_Pos_InnerRail.Error) AND (NOT GVL_1.Move_To_Pos_OuterRail.Error) THEN
				Inner_Rail.nAxisState:=standstill;
				Outer_Rail.nAxisState:=standstill;
            	GVL_1.Reset := FALSE;           // Clear reset command
				GVL_1.Machine_In_Error:=FALSE;
            	GVL_1.enStepBoot := 0;    // Restart boot sequence
     		END_IF
    	END_IF

		
	
	
END_CASE

GVL_1.Current_Pos_Inner:=LREAL_TO_INT(Inner_Rail.fActPosition);
GVL_1.Current_Pos_Outer:=LREAL_TO_INT(Outer_Rail.fActPosition);

END_PROGRAM

// Device/Application/Progs_In_Apollo/Machine State/Set_Parameter_Prog
PROGRAM Set_Parameter_Prog
VAR
END_VAR

IF GVL_1.Set_Parameters_Default THEN
	
//-------------------------------------------------------------------------------------------------	
	//Positions
	Parameters.ReadyPos_Inner:=1120;
	Parameters.ReadyPos_Outer:=1250;
	
	Parameters.Pick_Pos_Inner_Test_Prod:=10;
	Parameters.Pick_Pos_Outer_Test_Prod:=110;
	
	Parameters.Drop_Pos_Inner_Test_Prod:=1000;
	Parameters.Drop_Pos_Outer_Test_Prod:=1250;
	
	//dynamics
	Parameters.Speed_Test_Prod:=30;
	Parameters.ACC_DEC_Test_Prod:=1000;
	Parameters.Jerk_Prod:=100000;
	
	
	//distances
	Parameters.Distance_Move_After_PHC:=20;
	
	//Delays
	Parameters.Delay_Blow_Vacuum:=200;
	Parameters.Delay_Gripper_Closed_Before_Moving:=300;
	Parameters.Delay_Move_Conveyor_After_PHC_Covered:=1500;
	
	//Ventilator
	Parameters.Ventilator_Strength:=27649;
	
	//Wait times
	Parameters.Wait_Time_NoBatch:=5000;
	
	//Settings
	Parameters.Conveyor_Speed_Pick:=3;
	Parameters.Conveyor_Speed_Drop:=4;
//-------------------------------------------------------------------------------------------------	
	GVL_1.Set_Parameters_Default:=FALSE;
END_IF

END_PROGRAM

// Device/Application/Progs_In_Apollo/Test_Mode/Test_Full_Prod
PROGRAM Test_Full_Prod
VAR
	FB_Gripper:FunctionBlock_Gripper_Grip;
	FB_Dropping:FunctionBlock_Gripper_Drop;
	FB_Moving:FunctionBlock_Move_To_Pos;
	FB_ConveyorPick_Move:FunctionBlock_Move_Pick_Conveyor;
	
	Timer_AI:TON;
	Timer_Dropbox_Opened:TON;
	Timer_Open_Gripper_During_Drop:TON;
	Timer_Blow_Out:TON;
END_VAR

CASE GVL_1.enStepTestProd OF
	0: // wait until init
		(*
		IF NOT GVL_1.Machine_TestProd_Mode AND GVL_1.Start_production_Button THEN
			GVL_1.Cylinder_DropBox:=TRUE;
			Timer_Dropbox_Opened(IN:=TRUE,PT:=INT_TO_TIME(Parameters.Delay_DropBox_Opened));
			
			IF Timer_Dropbox_Opened.Q THEN
				GVL_1.Cylinder_DropBox:=FALSE;
				FB_ConveyorPick_Move(Right:=TRUE,LEFT:=FALSE,Speed:=3,Time_Moving:=Parameters.Delay_Conveyor_Move_After_DropBox_Opened,Start:=TRUE);
				IF FB_ConveyorPick_Move.Done THEN
					FB_ConveyorPick_Move(Start:=FALSE);
					Timer_Dropbox_Opened(IN:=FALSE);
					GVL_1.Machine_TestProd_Mode:=TRUE;
				END_IF
			END_IF
			
		END_IF
	*)
		
		//Check Init
		IF GVL_1.Machine_Ready_To_Run AND GVL_1.Machine_TestProd_Mode THEN
			//set dynamics
			GVL_1.Move_To_Pos_InnerRail.Velocity:=Parameters.Speed_Test_Prod;
			GVL_1.Move_To_Pos_InnerRail.Acceleration:=Parameters.ACC_DEC_Test_Prod;
			GVL_1.Move_To_Pos_InnerRail.Deceleration:=Parameters.ACC_DEC_Test_Prod;
			GVL_1.Move_To_Pos_InnerRail.Jerk:=Parameters.Jerk_Test_Prod;
			
			GVL_1.Move_To_Pos_OuterRail.Velocity:=Parameters.Speed_Test_Prod;
			GVL_1.Move_To_Pos_OuterRail.Acceleration:=Parameters.ACC_DEC_Test_Prod;
			GVL_1.Move_To_Pos_OuterRail.Deceleration:=Parameters.ACC_DEC_Test_Prod;
			GVL_1.Move_To_Pos_OuterRail.Jerk:=Parameters.Jerk_Test_Prod;
			
			GVL_1.Ventilator:=Parameters.Ventilator_Strength;
			
			GVL_1.enStepTestProd:=GVL_1.enStepTestProd+10;
		END_IF
		
		IF NOT GVL_1.Machine_TestProd_Mode THEN
			GVL_1.Ventilator:=0;
		END_IF
		
	10://Move to Ready
		GVL_1.Move_To_Pos_InnerRail.Velocity:=Parameters.Speed_Test_Prod_Slow;
		GVL_1.Move_To_Pos_InnerRail.Acceleration:=Parameters.ACC_DEC_Test_Prod_Slow;
		GVL_1.Move_To_Pos_InnerRail.Deceleration:=Parameters.ACC_DEC_Test_Prod_Slow;
		GVL_1.Move_To_Pos_InnerRail.Jerk:=Parameters.Jerk_Test_prod_Slow;
				
		GVL_1.Move_To_Pos_OuterRail.Velocity:=Parameters.Speed_Test_Prod_Slow;
		GVL_1.Move_To_Pos_OuterRail.Acceleration:=Parameters.ACC_DEC_Test_Prod_Slow;
		GVL_1.Move_To_Pos_OuterRail.Deceleration:=Parameters.ACC_DEC_Test_Prod_Slow;
		GVL_1.Move_To_Pos_OuterRail.Jerk:=Parameters.Jerk_Test_prod_Slow;
		
		FB_Moving(Start:=TRUE,Position_Inner:=Parameters.ReadyPos_Inner,Position_Outer:=Parameters.ReadyPos_Outer);
		
		
		IF FB_Moving.Done THEN
			FB_Moving(Start:=FALSE);
			GVL_1.Move_To_Pos_InnerRail.Velocity:=Parameters.Speed_Test_Prod;
			GVL_1.Move_To_Pos_InnerRail.Acceleration:=Parameters.ACC_DEC_Test_Prod;
			GVL_1.Move_To_Pos_InnerRail.Deceleration:=Parameters.ACC_DEC_Test_Prod;
			GVL_1.Move_To_Pos_InnerRail.Jerk:=Parameters.Jerk_Test_Prod;
		
			GVL_1.Move_To_Pos_OuterRail.Velocity:=Parameters.Speed_Test_Prod;
			GVL_1.Move_To_Pos_OuterRail.Acceleration:=Parameters.ACC_DEC_Test_Prod;
			GVL_1.Move_To_Pos_OuterRail.Deceleration:=Parameters.ACC_DEC_Test_Prod;
			GVL_1.Move_To_Pos_OuterRail.Jerk:=Parameters.Jerk_Test_Prod;
			GVL_1.enStepTestProd:=GVL_1.enStepTestProd+5;
		END_IF
	

	15: // Start AI
		IF NOT GVL_1.AI_Done THEN
			GVL_1.AI_Start:=TRUE;
		END_IF
		
		IF GVL_1.AI_Done THEN
			GVL_1.AI_Start:=FALSE;
			GVL_1.enStepTestProd:=GVL_1.enStepTestProd+5;
		END_IF

	
	20:// Move to Pick And grip as well Check if AI needs to be used

		IF NOT FB_ConveyorPick_Move.Done THEN
			FB_ConveyorPick_Move(Left:=GVL_1.Conveyor_Pick_Move_Left,Right:=GVL_1.Conveyor_Pick_Move_Right,Speed:=Parameters.Conveyor_Speed_Pick,Time_Moving:=GVL_1.Conveyor_Pick_Time,Start:=TRUE);
		END_IF
		
		IF FB_ConveyorPick_Move.Done THEN
			FB_Moving(Position_Inner:=GVL_1.Pick_Pos_Inner,Position_Outer:=GVL_1.Pick_Pos_Outer,Start:=TRUE);
		END_IF
		

		IF GVL_1.PHC_Gripper THEN
			FB_Moving(Halt:=TRUE);
			IF FB_Moving.Done THEN
				FB_Gripper(Start:=TRUE);
				
				IF FB_Gripper.Done THEN
					FB_Moving.Start:=FALSE;
					GVL_1.AI_Start:=FALSE;
					GVL_1.AI_Done:=FALSE;
					FB_Moving(Start:=FALSE);
					FB_Gripper(Start:=FALSE);
					FB_ConveyorPick_Move(Start:=FALSE);
					GVL_1.enStepTestProd:=GVL_1.enStepTestProd+10;
				END_IF	
			END_IF
		ELSIF FB_Moving.Done AND NOT GVL_1.PHC_Gripper THEN
			FB_Gripper(Start:=TRUE);
			
			IF FB_Gripper.Done THEN
				FB_Moving(Start:=FALSE);
				FB_Gripper(Start:=FALSE);
				FB_ConveyorPick_Move(Start:=FALSE);
				GVL_1.AI_Start:=FALSE;
				GVL_1.AI_Done:=FALSE;
				GVL_1.enStepTestProd:=GVL_1.enStepTestProd+10;
			END_IF
			
		END_IF
		

		

		
	30: // Move To Ready
		FB_Moving(Position_Inner:=Parameters.ReadyPos_Inner,Position_Outer:=Parameters.ReadyPos_Outer,Start:=TRUE);

		IF FB_Moving.Done THEN
			FB_Moving(Start:=FALSE);
			
			GVL_1.enStepTestProd:=GVL_1.enStepTestProd+10;
		END_IF
	40://Move to Drop
	

	
	
		GVL_1.Conveyor_Drop_Speed_A:=TRUE;
		GVL_1.Conveyor_Drop_Reverse:=TRUE;
	
	
		IF NOT GVL_1.PieceOnDropConveyor THEN
			
			Timer_Open_Gripper_During_Drop(IN:=TRUE,PT:=INT_TO_TIME(Parameters.Delay_Gripper_Open_During_Drop));
		
			IF Timer_Open_Gripper_During_Drop.Q THEN
				GVL_1.Gripper:=FALSE;
				Timer_Blow_Out(IN:=TRUE,PT:=INT_TO_TIME(parameters.Delay_Blow));
				GVL_1.Blow_Out:=TRUE;
				IF Timer_Blow_Out.Q THEN
					GVL_1.Blow_Out:=FALSE;
				END_IF
			END_IF
			
			GVL_1.Move_To_Pos_InnerRail(Axis:=Inner_Rail,Position:=Parameters.Drop_Pos_Inner_Test_Prod,Velocity:=Parameters.Speed_Test_Prod_Slow,Acceleration:=Parameters.ACC_DEC_Test_Prod_Slow,Deceleration:=Parameters.ACC_DEC_Test_Prod_Slow,Jerk:=Parameters.Jerk_Test_prod_Slow,Execute:=TRUE);
			GVL_1.Move_To_Pos_OuterRail(Axis:=Outer_Rail,Position:=Parameters.Drop_Pos_Outer_Test_Prod,Velocity:=Parameters.Speed_Test_Prod_Slow,Acceleration:=Parameters.ACC_DEC_Test_Prod_Slow,Deceleration:=Parameters.ACC_DEC_Test_Prod_Slow,Jerk:=Parameters.Jerk_Test_prod_Slow,Execute:=TRUE);
		END_IF
	

		
		IF GVL_1.Move_To_Pos_InnerRail.Done AND GVL_1.Move_To_Pos_OuterRail.Done THEN
			FB_Dropping(Start:=TRUE,Delay_Moving_After_Dropping:=Parameters.Delay_Move_After_Piece_Dropped);
			
			IF FB_Dropping.Done AND Timer_Blow_Out.Q THEN
				GVL_1.Conveyor_Drop_Speed_A:=FALSE;
				GVL_1.Conveyor_Drop_Reverse:=FALSE;
				FB_Dropping(Start:=FALSE);
				GVL_1.Move_To_Pos_InnerRail(Axis:=Inner_Rail,Execute:=FALSE);
				GVL_1.Move_To_Pos_OuterRail(Axis:=Outer_Rail,Execute:=FALSE);
				GVL_1.PieceOnDropConveyor:=TRUE;

				Timer_Open_Gripper_During_Drop(IN:=FALSE);
				Timer_Blow_Out(IN:=FALSE);
				GVL_1.enStepTestProd:=GVL_1.enStepTestProd+10;
			END_IF

		END_IF
		
	50:// Go to Ready
		

	
		GVL_1.Move_To_Pos_InnerRail(Axis:=Inner_Rail,Position:=Parameters.ReadyPos_Inner,Velocity:=Parameters.Speed_Test_Prod_Slow,Acceleration:=Parameters.ACC_DEC_Test_Prod_Slow,Deceleration:=Parameters.ACC_DEC_Test_Prod_Slow,Jerk:=Parameters.Jerk_Test_prod_Slow,Execute:=TRUE);
		GVL_1.Move_To_Pos_OuterRail(Axis:=Outer_Rail,Position:=Parameters.ReadyPos_Outer,Velocity:=Parameters.Speed_Test_Prod_Slow,Acceleration:=Parameters.ACC_DEC_Test_Prod_Slow,Deceleration:=Parameters.ACC_DEC_Test_Prod_Slow,Jerk:=Parameters.Jerk_Test_prod_Slow,Execute:=TRUE);
		GVL_1.PHC_Gripper:=FALSE;
		
		IF GVL_1.AI_Done THEN
			GVL_1.AI_Start:=FALSE;
			FB_ConveyorPick_Move(Left:=GVL_1.Conveyor_Pick_Move_Left,Right:=GVL_1.Conveyor_Pick_Move_Right,Speed:=Parameters.Conveyor_Speed_Pick,Time_Moving:=GVL_1.Conveyor_Pick_Time,Start:=TRUE);
		END_IF	
	
		IF GVL_1.Move_To_Pos_InnerRail.Done AND GVL_1.Move_To_Pos_OuterRail.Done THEN
			GVL_1.AI_Start:=TRUE;
			GVL_1.Move_To_Pos_InnerRail(Axis:=Inner_Rail,Execute:=FALSE);
			GVL_1.Move_To_Pos_OuterRail(Axis:=Outer_Rail,Execute:=FALSE);
			
			IF GVL_1.AI_Done THEN
				GVL_1.AI_Start:=FALSE;
				FB_ConveyorPick_Move(Left:=GVL_1.Conveyor_Pick_Move_Left,Right:=GVL_1.Conveyor_Pick_Move_Right,Speed:=Parameters.Conveyor_Speed_Pick,Time_Moving:=GVL_1.Conveyor_Pick_Time,Start:=TRUE);
			END_IF	
			
			GVL_1.enStepTestProd:=0;
		END_IF
		
		
		
END_CASE

END_PROGRAM

// Device/Application/Progs_In_Apollo/FunctionBlocks/FunctionBlock_Gripper_Grip
FUNCTION_BLOCK FunctionBlock_Gripper_Grip
VAR_INPUT
	Start:BOOL;
	
END_VAR
VAR_OUTPUT
	Done:BOOL;
END_VAR
VAR
	Timer_Grip:TON;
	Timer_Blow:TON;
END_VAR

CASE GVL_1.enFBGripping OF
	0: // Wait until Start
		IF Start AND NOT Done THEN
			GVL_1.enFBGripping:=GVL_1.enFBGripping+10;
		END_IF
		
		IF NOT Start THEN
			Done:=FALSE;
		END_IF
	
	10: // Grip and wait until done
		
	
	
	
		GVL_1.VacuumBlow:=TRUE;
		Timer_Blow(IN:=TRUE,PT:=INT_TO_TIME(Parameters.Delay_Blow_Vacuum));
		Timer_Grip(IN:=TRUE,PT:=INT_TO_TIME(Parameters.Delay_Gripper_Closed_Before_Moving));
		
		IF Timer_Blow.Q THEN
			GVL_1.VacuumBlow:=FALSE;
		END_IF
		
		IF Timer_Grip.Q THEN
			GVL_1.Gripper:=TRUE;
		END_IF
		
		IF Timer_Blow.Q AND Timer_Grip.Q THEN
			Timer_Blow(IN:=FALSE);
			Timer_Grip(IN:=FALSE);
			Done:=TRUE;
			GVL_1.enFBGripping:=0;
		END_IF
		


END_CASE

END_FUNCTION_BLOCK

// Device/Application/Progs_In_Apollo/FunctionBlocks/FunctionBlock_Gripper_Drop
FUNCTION_BLOCK FunctionBlock_Gripper_Drop
VAR_INPUT
	Start:BOOL;
	Delay_Moving_After_Dropping:INT;
END_VAR
VAR_OUTPUT
	Done:BOOL;
END_VAR
VAR
	Timer:TON;
	Timer_2:TON;
END_VAR

CASE GVL_1.enFBDropping OF
	0:// wait until init
		IF Start AND NOT Done THEN
			GVL_1.enFBDropping:=GVL_1.enFBDropping+10;
		END_IF
		
		IF NOT Start THEN
			Done:=FALSE;
		END_IF
	10:// Drop
		GVL_1.Gripper:=FALSE;
		//GVL_1.Blow_Out:=TRUE;
		Timer(IN:=TRUE,PT:=INT_TO_TIME(Delay_Moving_After_Dropping));
		
		//Timer_2(IN:=TRUE,PT:=INT_TO_TIME(parameters.Delay_Blow));
		
		IF Timer.Q THEN
			Timer(IN:=FALSE);
			//Timer_2(IN:=FALSE);
			Done:=TRUE;
			//GVL_1.Blow_Out:=FALSE;
			GVL_1.enFBDropping:=0;
		END_IF
END_CASE

END_FUNCTION_BLOCK

// Device/Application/Prog_In_DEV/Programms/Dropconveyor
PROGRAM Dropconveyor
VAR
	Timer:TON;
	Timer_2:TON;

END_VAR

CASE GVL_1.enStepDrop OF
	0:// Wait until piece on drop conveyor
		IF GVL_1.PieceOnDropConveyor THEN
			GVL_1.enStepDrop:=GVL_1.enStepDrop+10;
		END_IF
	10: // Wait until PHC is covered
		Timer_2(IN:=TRUE,PT:=INT_TO_TIME(Parameters.Wait_Time_Piece_Drop_Conveyor));
		GVL_1.Conveyor_Drop_Reverse:=TRUE;
		IF Parameters.Conveyor_Speed_Drop = 1 THEN
			GVL_1.Conveyor_Drop_Speed_C:=TRUE;
		ELSIF Parameters.Conveyor_Speed_Drop  = 2 THEN
			GVL_1.Conveyor_Drop_Speed_B:=TRUE;
		ELSIF Parameters.Conveyor_Speed_Drop  = 3 THEN
			GVL_1.Conveyor_Drop_Speed_A:=TRUE;
		ELSIF Parameters.Conveyor_Speed_Drop  = 4 THEN
			GVL_1.Conveyor_Drop_Speed_C:=TRUE;
			GVL_1.Conveyor_Drop_Speed_B:=TRUE;
		ELSIF Parameters.Conveyor_Speed_Drop =5 THEN
			GVL_1.Conveyor_Drop_Speed_A:=TRUE;
			GVL_1.Conveyor_Drop_Speed_B:=TRUE;
			GVL_1.Conveyor_Drop_Speed_C:=TRUE;
		END_IF
				
		
	
		IF GVL_1.PHC_Drop_Conveyor THEN
			GVL_1.enStepDrop:=GVL_1.enStepDrop+10;
		ELSIF Timer_2.Q THEN
			GVL_1.enStepDrop:=GVL_1.enStepDrop+10;
		END_IF
	20: // wait until PHC is not covered anymore
		IF NOT GVL_1.PHC_Drop_Conveyor THEN
			Timer(IN:=TRUE,PT:=INT_TO_TIME(parameters.Delay_Move_Conveyor_After_PHC_Covered));
			
			IF Timer.Q THEN
				GVL_1.Conveyor_Drop_Speed_A:=FALSE;
				GVL_1.Conveyor_Drop_Speed_B:=FALSE;
				GVL_1.Conveyor_Drop_Speed_C:=FALSE;
				GVL_1.Conveyor_Drop_Reverse:=FALSE;
				GVL_1.PieceOnDropConveyor:=FALSE;
				Timer(IN:=FALSE);
				Timer_2(IN:=FALSE);
				GVL_1.enStepDrop:=0;
			END_IF
			
		END_IF
END_CASE

END_PROGRAM

// Device/Application/PLC_PRG
PROGRAM PLC_PRG
VAR
END_VAR

END_PROGRAM

// Device/Application/Old_Progs/Apollo_Machine_State
PROGRAM Apollo_Machine_State
VAR

END_VAR

CASE GVL_1.enStepBoot OF
	0: // Check state of machine for booting. Machine now in turn_off state
		IF GVL_1.Turn_On AND NOT GVL_1.Machine_In_Error THEN
			GVL_1.enStepBoot:=GVL_1.enStepBoot+10;
		END_IF
		
		GVL_1.enStepTest:=0;
		
		GVL_1.Power_Drive_InnerRail(Axis:=Inner_Rail, Enable:=FALSE);
		GVL_1.Power_Drive_OuterRail(Axis:=Outer_Rail, Enable:=FALSE);
		
		GVL_1.Machine_Ready_To_Run:=FALSE;
		GVL_1.Turn_Off:=TRUE;
		
	10: // Boot up Drives 
		GVL_1.Turn_Off:=FALSE;
		
		GVL_1.Power_Drive_InnerRail(Axis:=Inner_Rail,Enable:=TRUE, bRegulatorOn:=TRUE, bDriveStart:=TRUE);
		GVL_1.Power_Drive_OuterRail(Axis:=Outer_Rail,Enable:=TRUE, bRegulatorOn:=TRUE, bDriveStart:=TRUE);
		

		
		IF GVL_1.Power_Drive_InnerRail.Status AND GVL_1.Power_Drive_OuterRail.Status THEN
			GVL_1.enStepBoot:=GVL_1.enStepBoot+10;
		END_IF
	20: // Robot ready to move
		GVL_1.Machine_Ready_To_Run:=TRUE;
END_CASE
//-------------------------------------------------------------------------------------------------	
//Error Handling
IF (GVL_1.Move_To_Pos_InnerRail.Error OR GVL_1.Move_To_Pos_OuterRail.Error) AND GVL_1.enStepBoot > 10 THEN
    GVL_1.Machine_In_Error := TRUE;
    GVL_1.Machine_Ready_To_Run := FALSE;
	
	GVL_1.enStepTest:=0;

    // Stop the Move Function Blocks by resetting Execute signals
    GVL_1.Move_To_Pos_InnerRail.Execute := FALSE;
    GVL_1.Move_To_Pos_OuterRail.Execute := FALSE;
ELSE
    GVL_1.Machine_In_Error := FALSE;
END_IF

// Reset Inner Rail if in error and reset button is pressed
IF GVL_1.Move_To_Pos_InnerRail.Error AND NOT GVL_1.Reset_InnerRail.Busy AND GVL_1.Reset THEN
    GVL_1.Reset_InnerRail(Axis := Inner_Rail, Execute := TRUE);
END_IF

// Reset Outer Rail if in error and reset button is pressed
IF GVL_1.Move_To_Pos_OuterRail.Error AND NOT GVL_1.Reset_OuterRail.Busy AND GVL_1.Reset THEN
    GVL_1.Reset_OuterRail(Axis := Outer_Rail, Execute := TRUE);
END_IF

// Once the reset is done, stop executing the reset function
IF GVL_1.Reset_InnerRail.Done THEN
    GVL_1.Reset_InnerRail(Axis := Inner_Rail, Execute := FALSE);
END_IF

IF GVL_1.Reset_OuterRail.Done THEN
    GVL_1.Reset_OuterRail(Axis := Outer_Rail, Execute := FALSE);
END_IF

//-------------------------------------------------------------------------------------------------	
//Power Handling
IF GVL_1.Turn_Off AND NOT GVL_1.Turn_On AND GVL_1.enStepBoot>0 THEN
	GVL_1.enStepTest:=0;
	GVL_1.Power_Drive_InnerRail(Axis:=Inner_Rail,Enable:=FALSE, bRegulatorOn:=FALSE, bDriveStart:=FALSE);
	GVL_1.Power_Drive_OuterRail(Axis:=Outer_Rail,Enable:=FALSE, bRegulatorOn:=FALSE, bDriveStart:=FALSE);
	GVL_1.enStepBoot:=0;
END_IF


//-------------------------------------------------------------------------------------------------	
//Positions reading
GVL_1.Current_Pos_Inner:=LREAL_TO_INT(Inner_Rail.fActPosition);
GVL_1.Current_Pos_Outer:=LREAL_TO_INT(Outer_Rail.fActPosition);

END_PROGRAM

// Device/Application/Old_Progs/FunctionBlock_Move_Guiders_Apollo
FUNCTION_BLOCK FunctionBlock_Move_Guiders_Apollo
VAR_INPUT
	Inner_Pos:INT;
	Outer_Pos:INT;
	Speed:INT;
	Acc_Dec:INT;
	Jk:INT; // jerk
	Start:BOOL;	
END_VAR
VAR_OUTPUT
	Done:BOOL;
END_VAR
VAR
END_VAR

CASE GVL_1.enFBMoveGuider OF
	0:// Wait until declaration
		IF Start AND NOT Done THEN
			GVL_1.enFBMoveGuider:=GVL_1.enFBMoveGuider+10;
		END_IF
		
	10: // Move to positions
		GVL_1.Move_To_Pos_InnerRail(Axis:=Inner_Rail,Position:=INT_TO_LREAL(Inner_Pos), Velocity:=INT_TO_LREAL(Speed), Acceleration:=INT_TO_LREAL(Acc_Dec),Deceleration:=INT_TO_LREAL(Acc_Dec),Jerk:=Jk, Execute:=TRUE);
		GVL_1.Move_To_Pos_OuterRail(Axis:=Outer_Rail,Position:=INT_TO_LREAL(Outer_Pos),Velocity:=INT_TO_LREAL(Speed),Acceleration:=INT_TO_LREAL(Acc_Dec),Deceleration:=INT_TO_LREAL(Acc_Dec),Jerk:=Jk, Execute:=TRUE);
		
		IF GVL_1.Move_To_Pos_InnerRail.Done AND GVL_1.Move_To_Pos_OuterRail.Done THEN
			GVL_1.enFBMoveGuider:=GVL_1.enFBMoveGuider+10;
		END_IF
		
	20: // reset moves and set done
		GVL_1.Move_To_Pos_InnerRail(Execute:=FALSE,Axis:=Inner_Rail);
		GVL_1.Move_To_Pos_OuterRail(Execute:=FALSE,Axis:=Outer_Rail);
		
		Done:=TRUE;
		
		GVL_1.enFBMoveGuider:=0;
END_CASE 

IF NOT Start THEN
	Done:=FALSE;
	GVL_1.enFBMoveGuider:=0;
END_IF

END_FUNCTION_BLOCK

// Device/Application/Old_Progs/Apollo_Running_Guiders_AND_PickConveyor
PROGRAM Apollo_Running_Guiders_AND_PickConveyor
VAR
	FB_Guider_Move:FunctionBlock_Move_Guiders_Apollo;
	FB_Conveyor_Move:FunctionBlock_Move_Pick_Conveyor;
	Difference_Move_Inner:INT;
	New_Pos_Inner:INT;
END_VAR

CASE GVL_1.enStepRun OF 
	0:// Wait until initialization
		IF GVL_1.Machine_Ready_To_Run AND GVL_1.Machine_Production_Mode THEN
			GVL_1.enStepRun:=GVL_1.enStepRun+10;
		END_IF
	10:// Check if batch is in machine
		IF GVL_1.PHC_PickConveyor_Front THEN
			GVL_1.NoBatchOnPickConveyor:=FALSE;
			GVL_1.enStepRun:=GVL_1.enStepRun+10;
		ELSE
			GVL_1.NoBatchOnPickConveyor:=TRUE;
		END_IF
	20: // Let Machine move to all necesseray pos for First AI detection
		FB_Guider_Move(Inner_Pos:=Parameters.ReadyPos_Inner,Outer_Pos:=Parameters.ReadyPos_Outer,Speed:=Parameters.Vel_Prod,Acc_Dec:=Parameters.Acc_Dec_Prod,Jk:=Parameters.Jerk_Prod,Start:=TRUE);
		
		GVL_1.Conveyor_Pick_Run:=TRUE;
		
		IF GVL_1.PHC_PickConveyor_END THEN
			GVL_1.Conveyor_Pick_Run:=FALSE;
		ELSIF GVL_1.PHC_PickConveyor_END AND FB_Guider_Move.Done THEN
			GVL_1.enStepRun:=GVL_1.enStepRun+5;
		END_IF
	25: // Reset
		FB_Guider_Move(Inner_Pos:=Parameters.ReadyPos_Inner,Outer_Pos:=Parameters.ReadyPos_Outer,Speed:=Parameters.Vel_Prod,Acc_Dec:=Parameters.Acc_Dec_Prod,Jk:=Parameters.Jerk_Prod,Start:=FALSE);
		
		GVL_1.enStepRun:=GVL_1.enStepRun+5;
	30: // Start AI
		GVL_1.AI_Start:=TRUE;
		
		IF GVL_1.AI_Done THEN
			GVL_1.enStepRun:=GVL_1.enStepRun+5;
		END_IF
	35: // reset
		GVL_1.AI_Start:=FALSE;
		GVL_1.AI_Done:=FALSE;
		
		GVL_1.enStepRun:=GVL_1.enStepRun+5;
	40: // Move Both Conveyor AND difference in Guider
		Difference_Move_Inner:=(GVL_1.Pick_Pos_Outer-GVL_1.Pick_Pos_Inner)-(Parameters.ReadyPos_Outer-Parameters.ReadyPos_Inner);
		New_Pos_Inner:=Parameters.ReadyPos_Inner-Difference_Move_Inner;
		
		FB_Guider_Move(Inner_Pos:=New_Pos_Inner,Outer_Pos:=Parameters.ReadyPos_Outer,Speed:=Parameters.Vel_Prod,Acc_Dec:=Parameters.Acc_Dec_Prod,Jk:=Parameters.Jerk_Prod,Start:=TRUE);
		FB_Conveyor_Move(Left:=GVL_1.Conveyor_Pick_Move_Left,Right:=GVL_1.Conveyor_Pick_Move_Right,Time_Moving:=GVL_1.Conveyor_Pick_Time,Start:=TRUE);
		
		IF FB_Guider_Move.Done AND FB_Conveyor_Move THEN
			GVL_1.enStepRun:=GVL_1.enStepRun+5;
		END_IF
	45: // Reset
		FB_Guider_Move(Inner_Pos:=New_Pos_Inner,Outer_Pos:=Parameters.ReadyPos_Outer,Speed:=Parameters.Vel_Prod,Acc_Dec:=Parameters.Acc_Dec_Prod,Jk:=Parameters.Jerk_Prod,Start:=FALSE);
		FB_Conveyor_Move(Left:=GVL_1.Conveyor_Pick_Move_Left,Right:=GVL_1.Conveyor_Pick_Move_Right,Time_Moving:=GVL_1.Conveyor_Pick_Time,Start:=FALSE);
		
		GVL_1.enStepRun:=GVL_1.enStepRun+5;
	50: // Go to Pick Pos
		FB_Guider_Move(Inner_Pos:=GVL_1.Pick_Pos_Inner,Outer_Pos:=GVL_1.Pick_Pos_Outer,Speed:=Parameters.Vel_Prod,Acc_Dec:=Parameters.Acc_Dec_Prod,Jk:=Parameters.Jerk_Prod,Start:=TRUE);
		
		IF FB_Guider_Move.Done THEN
			GVL_1.enStepRun:=GVL_1.enStepRun+5;
		
		END_IF
	55://Reset
		FB_Guider_Move(Inner_Pos:=GVL_1.Pick_Pos_Inner,Outer_Pos:=GVL_1.Pick_Pos_Outer,Speed:=Parameters.Vel_Prod,Acc_Dec:=Parameters.Acc_Dec_Prod,Jk:=Parameters.Jerk_Prod,Start:=TRUE);
		
		
 
		
		
		
		
		
END_CASE

END_PROGRAM

// Device/Application/Old_Progs/FunctionBlock_Move_Conveyor_Drop
FUNCTION_BLOCK FunctionBlock_Move_Conveyor_Drop
VAR_INPUT
END_VAR
VAR_OUTPUT
END_VAR
VAR
END_VAR

CASE GVL_1.enFBMoveConveyor_Drop OF
	0:// Init
		IF GVL_1.PieceOnDropConveyor THEN
			GVL_1.enFBMoveConveyor_Drop:=GVL_1.enFBMoveConveyor_Drop+10;
		END_IF
	10: // Wait until PHC is covered
		IF GVL_1.PHC_Drop_Conveyor THEN
			GVL_1.enFBMoveConveyor_Drop:=GVL_1.enFBMoveConveyor_Drop+10;
		END_IF
	20:// wait until PHC is not covered anymore 
END_CASE

END_FUNCTION_BLOCK

// Device/Application/Prog_In_DEV/Programms/Apollo_RunMode_Main
PROGRAM Apollo_RunMode_Main
VAR
	FB_MoveConvPick:FunctionBlock_Move_Pick_Conveyor;
	FB_MoveRobot:FunctionBlock_Move_To_Pos;
	FB_Grip:FunctionBlock_Gripper_Grip;
END_VAR

CASE GVL_1.enStepRun OF
	0: // INIT
		IF NOT GVL_1.Machine_In_Error AND GVL_1.Machine_Production_Mode AND GVL_1.BatchOnPickConveyor THEN
			//Set Dynamics
			GVL_1.Move_To_Pos_InnerRail.Velocity:=Parameters.Vel_Prod;
			GVL_1.Move_To_Pos_InnerRail.Acceleration:=Parameters.Acc_Dec_Prod;
			GVL_1.Move_To_Pos_InnerRail.Deceleration:=Parameters.Acc_Dec_Prod;
			GVL_1.Move_To_Pos_InnerRail.Jerk:=Parameters.Jerk_Prod;
			
			GVL_1.Move_To_Pos_OuterRail.Velocity:=Parameters.Vel_Prod;
			GVL_1.Move_To_Pos_OuterRail.Acceleration:=Parameters.Acc_Dec_Prod;
			GVL_1.Move_To_Pos_OuterRail.Deceleration:=Parameters.Acc_Dec_Prod;
			GVL_1.Move_To_Pos_OuterRail.Jerk:=Parameters.Jerk_Prod;
			
			GVL_1.enStepRun:=GVL_1.enStepRun+10;
		END_IF
		
		IF NOT GVL_1.BatchOnPickConveyor AND GVL_1.PutinBatch THEN
			GVL_1.BatchOnPickConveyor:=TRUE;
			GVL_1.PutinBatch:=FALSE;
		END_IF
		
		
	10:// Check if batch is in machine
		IF GVL_1.PHC_PickConveyor_Front OR GVL_1.PHC_PickConveyor_END OR GVL_1.AI_Done THEN
			GVL_1.BatchOnPickConveyor:=TRUE;
			FB_MoveConvPick(Start:=FALSE);
			GVL_1.enStepRun:=GVL_1.enStepRun+10;
		ELSE
			FB_MoveConvPick(Start:=TRUE,Right:=TRUE,Speed:=Parameters.Conveyor_Speed_Pick);
			IF FB_MoveConvPick.Done AND NOT (GVL_1.PHC_PickConveyor_Front OR GVL_1.PHC_PickConveyor_END) THEN
				GVL_1.BatchOnPickConveyor:=FALSE;
				GVL_1.enStepRun:=0;
			END_IF
		END_IF
		
		
	20:// Check if robot is in ready pos and if conveyor already moved in correct positions
		FB_MoveRobot(Position_Inner:=Parameters.ReadyPos_Inner,Position_Outer:=Parameters.ReadyPos_Outer,Start:=TRUE);

		IF FB_MoveRobot.Done THEN
			FB_MoveRobot(Start:=FALSE);
			GVL_1.enStepRun:=GVL_1.enStepRun+10;
		END_IF	

	30://Check if Positions are in memory. If no then do detection If yes continue
		IF NOT GVL_1.AI_Detection_Memory THEN
			GVL_1.AI_Start:=TRUE;
			
			IF GVL_1.AI_Done THEN
				
				GVL_1.AI_Start:=FALSE;
				GVL_1.AI_Done:=FALSE;
				GVL_1.enStepRun:=GVL_1.enStepRun+10;
			END_IF
		ELSE
			GVL_1.enStepRun:=GVL_1.enStepRun+10;
		END_IF
	40: // Move conveyor And pick 
		//Check if conveyor is already moved in correct position
		IF GVL_1.Conveyor_Movement_Memory THEN
			FB_MoveRobot(Position_Inner:=GVL_1.Pick_Pos_Inner,Position_Outer:=GVL_1.Pick_Pos_Outer,Start:=TRUE);
			IF FB_MoveRobot.Done THEN
				FB_MoveRobot(Start:=FALSE);
				GVL_1.Conveyor_Movement_Memory:=FALSE;
				GVL_1.enStepRun:=GVL_1.enStepRun+10;
			END_IF
		ELSE
			FB_MoveConvPick(Start:=TRUE,Left:=GVL_1.Conveyor_Pick_Move_Left,Right:=GVL_1.Conveyor_Pick_Move_Right,Speed:=Parameters.Conveyor_Speed_Pick,Time_Moving:=GVL_1.Conveyor_Pick_Time);
			IF FB_MoveConvPick.Done THEN
				FB_MoveRobot(Position_Inner:=GVL_1.Pick_Pos_Inner,Position_Outer:=GVL_1.Pick_Pos_Outer,Start:=TRUE);
				IF FB_MoveRobot.Done THEN
					FB_Grip(Start:=TRUE);
					IF FB_Grip.Done THEN
						FB_MoveConvPick(Start:=FALSE);
						FB_MoveRobot(Start:=FALSE);
						FB_Grip(Start:=FALSE);
					END_IF
				END_IF
			END_IF
		END_IF
	50: // Move to drop using path
		
		
		
		
END_CASE
FB_MoveConvPick();

END_PROGRAM

// Device/Application/Old_Progs/Apollo_Running_GuiderMovement
PROGRAM Apollo_Running_GuiderMovement
VAR
END_VAR

CASE GVL_1.enStepRunMove OF
	0:// Wait until initialization
		IF GVL_1.Machine_Ready_To_Run AND GVL_1.Machine_Production_Mode THEN
			GVL_1.enStepRun:=GVL_1.enStepRun+10;
		END_IF
	10: // Move To ReadyPos
		
END_CASE

END_PROGRAM

// Device/Application/Main_Page
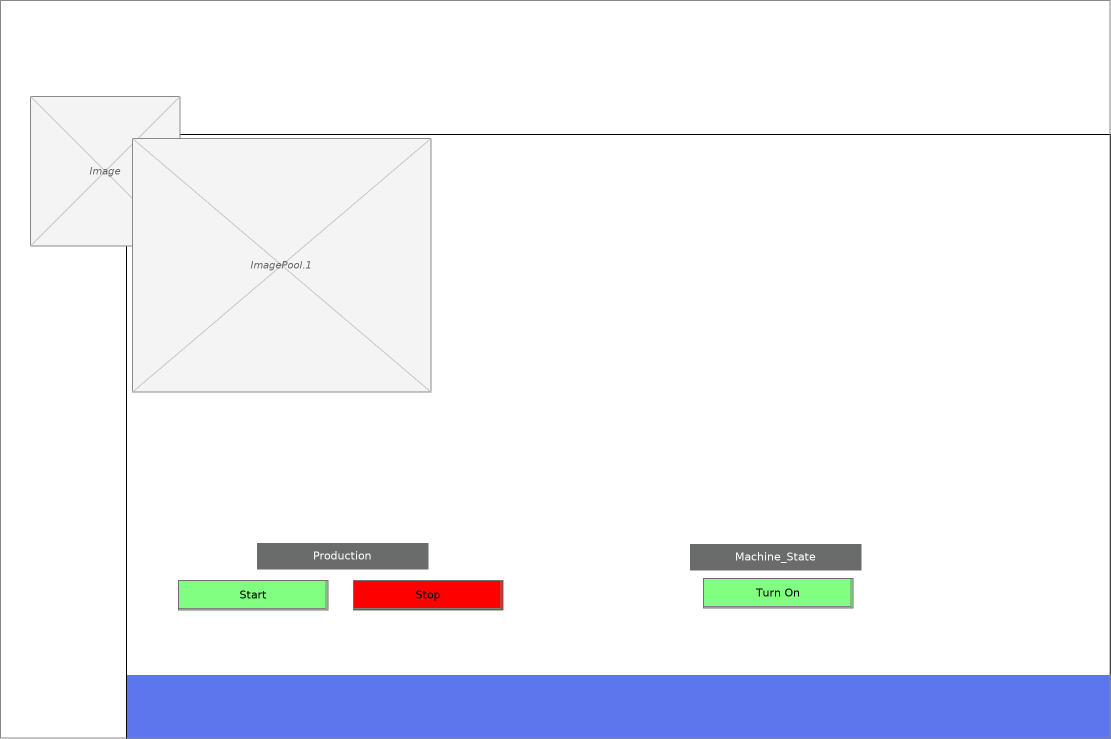
VISUALIZATION Main_Page  // 1111x739, background image 
    Rectangle (126,134 985x605)
    Button (178,580 150x30), "Start"
        tap GVL_1.Machine_TestProd_Mode p1329445385=TRUE
    Button (353,580 150x30), "Stop"
        tap GVL_1.Machine_TestProd_Mode
    Image (30,96 150x150)
    Image (132,138 299x254), image: ImagePool.1
    Rectangle (257,543 171x26), "Production"
    Rectangle (690,544 171x26), "Machine_State"
    Button (703,578 150x30), "Turn On"
        tap GVL_1.Turn_On
    Rectangle (127,675 984x64)
END_VISUALIZATION
